ABB RobotStudio station: Project4.rsstnx

Station Project4 (saved by RobotStudio 22.3.10141.1)
Controller Controlador1
  mechanical unit ROB_1: IRB120_3_58__01, 6 joints, base frame (0, 0, 0) mm
Layout (positions relative to the parent item):
  - IRB120_3_58__01 [mechanism, from Robots\IRB120_3_58_G_01.rslib] at (0, 0, 0) mm; joint values [-0.9924, -0.0465, -0.014, -0.5633, 1.3764, -6.9811] (rad or m)
  - Soldador [mechanism] at (133.6, -273.62, 589.08) mm, rotated rx -145.97 ry -9.91 rz 162.32 deg
      TCP Soldador at (0, 0, 110) mm
      links: Pieza_3
  - Pieza_1 [part], size 50 x 50 x 500 mm
Attachment: Soldador is attached to IRB120_3_58__01 / Link6
Targets, tools, work objects and paths stored in the station, written as RAPID:
! task T_ROB1
MODULE CalibData
  PERS tooldata Soldador:=[TRUE,[[0,0,110],[1,0,0,0]],[0.1,[0,0,10],[1,0,0,0],0,0,0]];
ENDMODULE

